KUKA KRL program: R2_Milling.src, R2_Milling.dat

--- R2_Milling.src ---
&ACCESS RV2
&REL 6
&PARAM DISKPATH = KRC:\R1\TP\Milling
DEF R2_Milling ( )
   BOOL lbOK
   ;FOLD INIT
      ;******************************************************************
      ;* Safety Monitoring                                              *
      ;******************************************************************
      $CYCFLAG[cycEmStop]       = NOT $ALARM_STOP OR NOT $MOVE_ENABLE
      ;******************************************************************
      ;* Enable Switch monitoring                                       *
      ;******************************************************************
      IF $T1 AND NOT $USER_SAF THEN
         gbSpindleStart = FALSE
      ENDIF
      ;******************************************************************
      ;* gbRobControlActive = FALSE always when Prog not Runnin         *
      ;******************************************************************
      IF($PRO_STATE1==#P_RESET) OR ($PRO_STATE1==#P_FREE) THEN
         gbRobControlActive = FALSE
      ELSE
         gbRobControlActive = TRUE
         gnSetSpindleSpeedHmi = 0
      ENDIF

      ;******************************************************************
      ;* Act Spindle speed monitoring for HMI                           *
      ;******************************************************************
      gnActSpindleSpeed = getActSpindleSpeed(gDISpindleActSpeed)
      ;******************************************************************
      ;* Spindle Runing state monitoring for HMI                        *
      ;******************************************************************

   ;ENDFOLD INIT
   ;FOLD CLAMP TOOL
      ;******************************************************************
      ;* Call Clamp/Unclamp program Based on HMI                        *
      ;* After clamping gbClampHmiEnable will be  FALSE (Automaticaly)  *
      ;******************************************************************
      IF (gbClampHmiEnable AND $T1 AND NOT gbRobControlActive)OR ($TIMER_STOP[gnHsdToolClamTimer] == FALSE) THEN
         IF ($TIMER_STOP[gnHsdToolClamTimer] == FALSE) THEN
            IF ($TIMER[gnHsdToolClamTimer] >= 2500)THEN
               $TIMER_STOP[gnHsdToolClamTimer] = TRUE
               $TIMER[gnHsdToolClamTimer] = 0
               gDOToolClamp        = FALSE
               gDOToolRelease      = FALSE
            ENDIF
         ENDIF
         IF gbSpindleClamp THEN
            SpindleClamp(TRUE)
         ENDIF
         IF gbSpindleRelease THEN
            SpindleClamp(FALSE)
         ENDIF
      ENDIF

   ;ENDFOLD CLAMP
   ;FOLD SPINDLE CONTROL
      ;******************************************************************
      ;* Main Spindle Run function                                      *
      ;* Start / Stop / QuickStop                                       *
      ;* Speed                                                          *
      ;* SpindleWord (Acel,Decel,Wait)                                  *
      ;******************************************************************
      ;IF $CYCFLAG[cycEmStop]  THEN
         ;oFreqconverterCtlw = gsSpindleWord.WaitForCommand
         ;oConverterSetSpeed = 0
         ;gISetSpeed = 0
         ;gbSpindleStart = FALSE
      ;ELSE
         oSpindleOperMode   = gnSpindleOperatinMode
         ;******************************************************************
         ;* Spindle Operated from Program                                  *
         ;******************************************************************
         lbOK =          NOT  gDi_HsdS2
         lbOK = lbOK     AND  gDi_HsdS1
         lbOK = lbOK     AND  gDi_HsdElFanRunning
         lbOK = lbOK AND NOT  gDi_HsdNoTool
         lbOK = lbOK     AND  gDi_HsdThermo

         IF lbOK THEN
            IF gbSpindleStart AND NOT gbRobControlActive THEN
               $TIMER_STOP[gnHsdStartTimer] = TRUE
               $TIMER[gnHsdStartTimer] = 0
               oConverterSetSpeed = getSpindleSpeed(gnSetSpindleSpeedHmi)
               oFreqconverterCtlw = gsSpindleWord.RunSpindle
               $TIMER_STOP[gnHsdStartTimer] = FALSE
            ENDIF
            ;******************************************************************
            ;* Spindle Operated from HMI                                      *
            ;******************************************************************
            IF gbSpindleStart AND gbRobControlActive THEN
               $TIMER_STOP[gnHsdStartTimer] = TRUE
               $TIMER[gnHsdStartTimer] = 0
               oConverterSetSpeed = getSpindleSpeed(gISetSpeed)
               oFreqconverterCtlw = gsSpindleWord.RunSpindle
               $TIMER_STOP[gnHsdStartTimer] = FALSE
            ENDIF
         ENDIF
         ;******************************************************************
         ;* Stop Spindle                                                   *
         ;******************************************************************
         IF (NOT gDI_HsdNotRunning AND NOT gbSpindleStart) OR NOT lbOK THEN
            oFreqconverterCtlw = gsSpindleWord.StopDec1
            $TIMER_STOP[gnHsdStartTimer] = TRUE
            $TIMER[gnHsdStartTimer] = 0
         ELSE
            ;******************************************************************
            ;*After Stop change controlWord to WAIT                           *
            ;******************************************************************
            IF  ($TIMER[gnHsdStartTimer] > 500) THEN
               $TIMER_STOP[gnHsdStartTimer] = TRUE
               $TIMER[gnHsdStartTimer] = 0
               oFreqconverterCtlw = gsSpindleWord.WaitForCommand
            ENDIF
         ENDIF
      ;;ENDIF
   ;ENDFOLD SPINDLE CONTROL
   ; FOLD CLAMP TABLE
      IF( NOT gbRobControlActive)THEN
         TableClamp(gbTableClamp)
      ENDIF
   ;ENDFOLD CLAMP TABLE
END

;FOLD getSpindleSpeed
   DEFFCT INT getSpindleSpeed (lnSetSpindleSpeed :IN)
      INT lnSetSpindleSpeed

      IF lnSetSpindleSpeed<0 THEN
         RETURN (lnSetSpindleSpeed/10+65535)
      ELSE
         RETURN (lnSetSpindleSpeed/10)
      ENDIF

      RETURN 0
   ENDFCT

;ENDFOLD getSpindleSpeed
;FOLD getActSpindleSpeed
   DEFFCT INT getActSpindleSpeed (lnSpeedFeedback :IN)
      INT lnSpeedFeedback
      IF lnSpeedFeedback>30000 THEN
         gbSpindleDirCw = FALSE
         gbSpindleDirCcw = TRUE
         RETURN  ((65535 - lnSpeedFeedback)*10)
      ELSE
         IF (lnSpeedFeedback>0) AND  (lnSpeedFeedback<30000) THEN
            gbSpindleDirCw = TRUE
            gbSpindleDirCcw = FALSE
            RETURN (lnSpeedFeedback*10)
         ELSE
            gbSpindleDirCw = FALSE
            gbSpindleDirCcw = FALSE
         ENDIF
      ENDIF
      RETURN 0
   ENDFCT

;ENDFOLD getActSpindleSpeed
;FOLD SpindleRun
   GLOBAL DEF SpindleRun (lbStartSpindle :IN,lrSpindleRPM :IN, FI_DIRECTION:IN)
      BOOL lbStartSpindle
      INT lrSpindleRPM
      DECL TYPMillDirection FI_DIRECTION
      IF lbStartSpindle THEN
         SWITCH FI_DIRECTION
            CASE #CLOCKWISE
               gISetSpeed = -lrSpindleRPM
            CASE #COUNTERCLOCKWISE
               gISetSpeed = lrSpindleRPM
            DEFAULT
         ENDSWITCH
         gbSpindleStart = TRUE
      ELSE
         gbSpindleStart = FALSE
      ENDIF

   END

;ENDFOLD SpindleRun
;FOLD SpindleClamp
   GLOBAL DEF SpindleClamp(lbToolReleaseReq :IN)
      BOOL lbToolReleaseReq

      IF  gDI_HsdNotRunning THEN
         IF NOT lbToolReleaseReq AND $TIMER_STOP[gnHsdToolClamTimer] THEN
            $TIMER[gnHsdToolClamTimer] = 0
            $TIMER_STOP[gnHsdToolClamTimer] = FALSE
            gDOToolClamp        = TRUE
            gDOToolRelease      = FALSE
         ENDIF
         IF lbToolReleaseReq AND $TIMER_STOP[gnHsdToolClamTimer] THEN
            $TIMER[gnHsdToolClamTimer] = 0
            $TIMER_STOP[gnHsdToolClamTimer] = FALSE
            gDOToolClamp        = FALSE
            gDOToolRelease      = TRUE
            gbClampHmiEnable    = FALSE
         ENDIF
      ENDIF

   END

;ENDFOLD SpindleClamp

DEF TableClamp(lbValue :IN)
   BOOL lbValue

   gO_Clamp_1 = lbValue
   gO_UnClamp_1 = NOT lbValue
   gO_Clamp_2 = lbValue
   gO_UnClamp_2 = NOT lbValue
END

--- R2_Milling.dat ---
&ACCESS RV2
&REL 6
&PARAM DISKPATH = KRC:\R1\TP\Milling
DEFDAT  R2_MILLING PUBLIC

GLOBAL CONST INT gnHsdToolClamTimer=34
GLOBAL CONST INT gnHsdStartTimer=33



GLOBAL SIGNAL gDi_HsdS2 $IN[1535]
GLOBAL SIGNAL gDi_HsdS1 $IN[1536]
GLOBAL SIGNAL gDi_HsdS3 $IN[1537]
GLOBAL SIGNAL gDi_HsdElFanRunning $IN[1538]
GLOBAL SIGNAL gDi_HsdElecOk $IN[1539]
GLOBAL SIGNAL gDi_HsdNoTool $IN[1540]
GLOBAL SIGNAL gDi_HsdThermo $IN[1541]
GLOBAL SIGNAL gDI_HsdNotRunning $IN[1542]



GLOBAL SIGNAL gDOToolRelease $OUT[1536]
GLOBAL SIGNAL gDIToolReleasedOK $IN[125]
GLOBAL SIGNAL gDOToolClamp $OUT[1537]

GLOBAL SIGNAL gO_Clamp_1 $OUT[1531]
GLOBAL SIGNAL gO_UnClamp_1 $OUT[1532]
GLOBAL SIGNAL gO_Clamp_2 $OUT[1533]
GLOBAL SIGNAL gO_UnClamp_2 $OUT[1534]

GLOBAL SIGNAL gDISpindleActSpeed $IN[224]  TO $IN[239]
GLOBAL SIGNAL gDISpindleEnableOK $IN[161]
GLOBAL SIGNAL iConverterStatus $IN[208]  TO $IN[223]

GLOBAL SIGNAL oFreqconverterCtlw $OUT[101]  TO $OUT[116] ; instead of cw in sps
GLOBAL SIGNAL oSpindleOperMode $OUT[117]  TO $OUT[124]
GLOBAL SIGNAL oConverterSetSpeed $OUT[601]  TO $OUT[616]
GLOBAL SIGNAL gDOSpindleEnable $OUT[133]


DECL GLOBAL BOOL gbSpindleStart=FALSE
DECL GLOBAL BOOL gbTooleReleaseReq=FALSE
DECL GLOBAL INT gnSpindleOperatinMode=2


GLOBAL STRUC sSpindleWord INT RunSpindle,StopDec1,QuickStop,WaitForCommand
DECL GLOBAL sSpindleWord gsSpindleWord={RunSpindle 127,StopDec1 128,QuickStop 129,WaitForCommand 126}

GLOBAL INT gISetSpeed=-10450
GLOBAL INT gIActSpeed=-8000
GLOBAL INT giSpindlespeedchecksum=-800
GLOBAL BOOL gbRobControlActive=FALSE
GLOBAL BOOL gbRobControlEnable=FALSE
GLOBAL BOOL gbRobControlRequest=FALSE
GLOBAL BOOL gbMillSystemWarning=FALSE
GLOBAL BOOL gbDirectionClockwise=TRUE
GLOBAL INT cycEmStop=30
GLOBAL INT oMinSpindleRpm=0
GLOBAL INT oMaxSpindleRpm=15000
GLOBAL INT gnActSpindleSpeed=0
GLOBAL INT gnSetSpindleSpeedHmi=0
GLOBAL BOOL gbSpindleDirCcw=FALSE
GLOBAL BOOL gbSpindleDirCw=FALSE
GLOBAL BOOL gbClampHmiEnable=FALSE
GLOBAL BOOL gbSpindleClamp=FALSE
GLOBAL BOOL gbSpindleRelease=FALSE
GLOBAL BOOL gbTableClamp=TRUE
GLOBAL BOOL gbSpindleBlowOff=FALSE
GLOBAL BOOL gbToolClampCheckReq=FALSE


GLOBAL ENUM TYPMillDirection CLOCKWISE,COUNTERCLOCKWISE
GLOBAL STRUC sR2Param REAL VC,FZ,AP,Dia,NrE,RPM,rSpeed,FRAME toolOffset
DECL GLOBAL sR2Param gsR2Param[16]
gsR2Param[1]={VC 0.100000,FZ 0.200000,AP 0.300000,Dia 24.0000,NrE 3.00000,toolOffset {X 0.0,Y 0.0,Z 0.0,A 0.0,B 0.0,C 0.0}}


ENDDAT
